SYSTEM NewBlockTestProject
  (* Version 1.0, 2025-07-09, dakudryashev *)
  APPLICATION NewBlockTestProjectApp
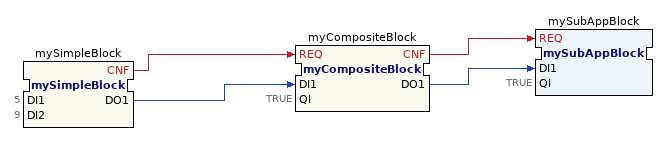
    FBS
      mySimpleBlock : mySimpleBlock(DI1 := 5, DI2 := 9);
      myCompositeBlock : myCompositeBlock(QI := TRUE);
    END_FBS
    SUBAPPS
      mySubAppBlock : mySubAppBlock(QI := TRUE);
    END_SUBAPPS
    EVENT_CONNECTIONS
      mySimpleBlock.CNF TO myCompositeBlock.REQ;
      myCompositeBlock.CNF TO mySubAppBlock.REQ;
    END_CONNECTIONS
    DATA_CONNECTIONS
      mySimpleBlock.DO1 TO myCompositeBlock.DI1;
      myCompositeBlock.DO1 TO mySubAppBlock.DI1;
    END_CONNECTIONS
  END_APPLICATION
  DEVICE FORTE_PC : FORTE_PC(MGR_ID := "localhost:61499" (* Device manager socket ID *))
    {SET_ATTRIBUTE(Profile, HOLOBLOC)}
    RESOURCE EMB_RES : EMB_RES
      EVENT_CONNECTIONS
        START.COLD TO NewBlockTestProjectApp.mySimpleBlock.REQ;
      END_CONNECTIONS
    END_RESOURCE
  END_DEVICE
  MAPPINGS
    NewBlockTestProjectApp.mySimpleBlock ON FORTE_PC.EMB_RES;
    NewBlockTestProjectApp.mySubAppBlock ON FORTE_PC.EMB_RES;
    NewBlockTestProjectApp.myCompositeBlock ON FORTE_PC.EMB_RES;
  END_MAPPINGS
  SEGMENTS
    Ethernet : Ethernet;
  END_SEGMENTS
  LINKS
    FORTE_PC => Ethernet;
  END_LINKS
END_SYSTEM
